{attribute 'call_after_init'}
FUNCTION_BLOCK FB_AnyToString_Test EXTENDS TcUnit.FB_TestSuite IMPLEMENTS TcUnit.I_RunnableTestSuite
VAR
    Assert : TcUnit.FB_Assert;
END_VAR

METHOD FB_init : BOOL
VAR_INPUT
	bInitRetains : BOOL; // if TRUE, the retain variables are initialized (warm start / cold start)
	bInCopyCode : BOOL;  // if TRUE, the instance afterwards gets moved into the copy code (online change)
END_VAR
SUPER^.RegisterTestSuite(THIS^);
END_METHOD

METHOD RunTests : TCUNIT.E_TestSuiteRunState
Test_String();
Test_INT();
Test_REAL();

RunTests := TCUNIT.E_TestSuiteRunState.FINISHED;
END_METHOD

METHOD Test_INT
VAR
    expected: STRING(10);
    actual: STRING(10);
    
    testINT: INT;
END_VAR
TEST('Test_INT');

expected := '1001';

testINT := 1001;
actual := anyToString(testINT);

Assert.AssertEquals_STRING(expected, actual, 'Any INT does not match');
END_METHOD

METHOD Test_REAL
VAR
    expected: STRING(10);
    actual: STRING(10);
    
    testREAL: REAL;
END_VAR
TEST('Test_REAL');

expected := '13.789';

testREAL := 13.789;
actual := anyToString(testREAL);

Assert.AssertEquals_STRING(expected, actual, 'Any REAL does not match');
END_METHOD

METHOD Test_String
VAR
    expected: STRING(10);
    actual: STRING(10);
END_VAR
TEST('Test_String');

expected := 'hello';

actual := anyToString(expected);

Assert.AssertEquals_STRING(expected, actual, 'Any String does not match');
END_METHOD

END_FUNCTION_BLOCK

(* stored: Version 1.1.0.1, ProductVersion 3.1.4022.12
   POU FB_AnyToString_Test: Id {3d6f8082-9d38-427c-9d5d-52917f8cfb73}, SpecialFunc None
   Method FB_init: Id {266858c1-8e8e-421f-b6f9-ddd28c528a56}
   Method RunTests: Id {19565166-4ad0-41f6-88f3-8f5948776325}
   Method Test_INT: Id {8c6b2744-a841-4815-b23a-46518637b988}
   Method Test_REAL: Id {50a94e1f-8437-44df-94c8-77a8343e8805}
   Method Test_String: Id {89ba2d1b-5887-4e66-9fd6-4fafe26e4bc3} *)
